% RSLogix 500 project TEMPLATE_BAK000.RSS, saved by version 8.30.00.16 %
PROJECT "UNTITLED"    % processor: Bul.1763 MicroLogix 1100 Series B %

PROGRAM FILES
  LAD 2 "MAIN"  10 rungs
  LAD 3 "DIGIT IN"  2 rungs
  LAD 4 "DIGIT OUT"  2 rungs
  LAD 5 "CTRL LOGIC"  5 rungs
  LAD 6 "HOA"  5 rungs
  LAD 7 "ANLG IN"  2 rungs
  LAD 8 "ANLG OUT"  1 rungs
  LAD 9 "ALARMS"  5 rungs
  LAD 10 "SYS MODES"  1 rungs
  LAD 11 "PROC LOGIC"  1 rungs

DATA FILES
  O0 OUTPUT  4 elements
  I1 INPUT  6 elements
  S2 STATUS  66 elements
  B3 BINARY  1 elements
  T4 TIMER  1 elements
  C5 COUNTER  1 elements
  R6 CONTROL  1 elements
  N7 INTEGER  1 elements
  F8 FLOAT  1 elements

LADDER 2 "MAIN"
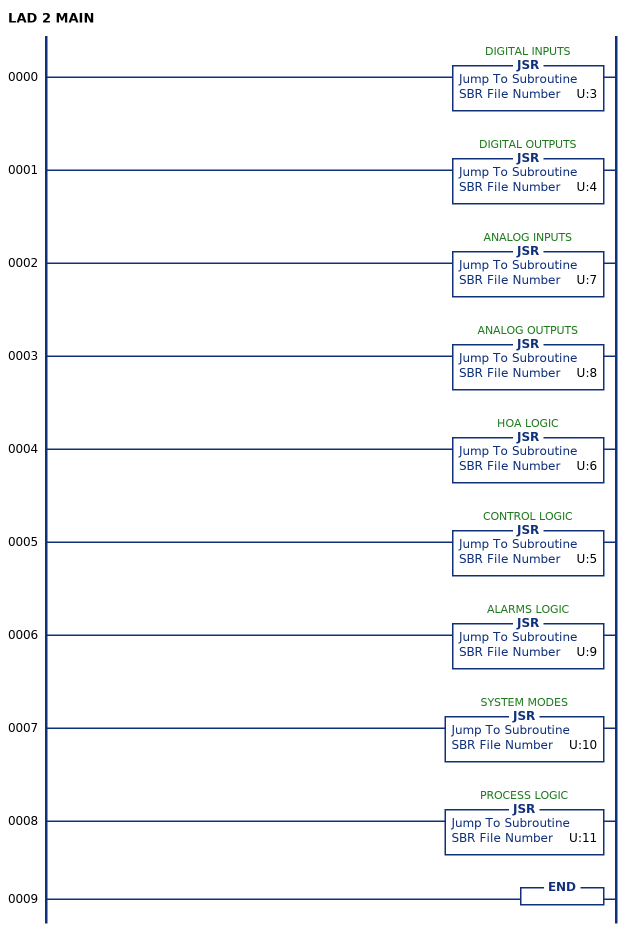
% Rung: 0 %
SOR JSR U:3 EOR
%   U:3  "DIGITAL INPUTS" %
% Rung: 1 %
SOR JSR U:4 EOR
%   U:4  "DIGITAL OUTPUTS" %
% Rung: 2 %
SOR JSR U:7 EOR
%   U:7  "ANALOG INPUTS" %
% Rung: 3 %
SOR JSR U:8 EOR
%   U:8  "ANALOG OUTPUTS" %
% Rung: 4 %
SOR JSR U:6 EOR
%   U:6  "HOA LOGIC" %
% Rung: 5 %
SOR JSR U:5 EOR
%   U:5  "CONTROL LOGIC" %
% Rung: 6 %
SOR JSR U:9 EOR
%   U:9  "ALARMS LOGIC" %
% Rung: 7 %
SOR JSR U:10 EOR
%   U:10  "SYSTEM MODES" %
% Rung: 8 %
SOR JSR U:11 EOR
%   U:11  "PROCESS LOGIC" %
% Rung: 9 %
SOR END EOR

LADDER 3 "DIGIT IN"
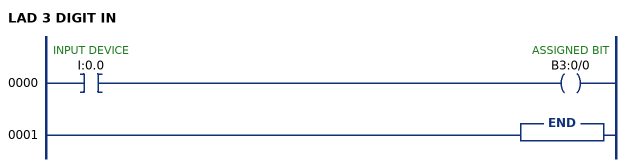
% Rung: 0 %  % edit flag set %
SOR XIC I:0.0 OTE B3:0/0 EOR
%   I:0.0  "INPUT DEVICE" %
%   B3:0/0  "ASSIGNED BIT" %
% Rung: 1 %
SOR END EOR

LADDER 4 "DIGIT OUT"
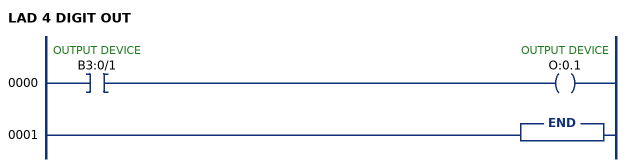
% Rung: 0 %  % edit flag set %
SOR XIC B3:0/1 OTE O:0.1 EOR
%   B3:0/1  "OUTPUT DEVICE" %
%   O:0.1  "OUTPUT DEVICE" %
% Rung: 1 %
SOR END EOR

LADDER 5 "CTRL LOGIC"
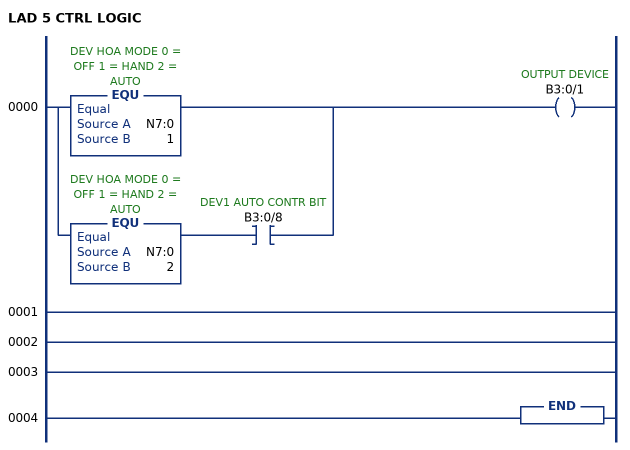
% Rung: 0 %  % edit flag set %
SOR BST EQU N7:0 1 NXB EQU N7:0 2 XIC B3:0/8 BND OTE B3:0/1 EOR
%   N7:0  "DEV HOA MODE 0 = OFF 1 = HAND 2 = AUTO" %
%   B3:0/8  "DEV1 AUTO CONTR BIT" %
%   B3:0/1  "OUTPUT DEVICE" %
% Rung: 1 %  % edit flag set %
SOR EOR
% Rung: 2 %  % edit flag set %
SOR EOR
% Rung: 3 %  % edit flag set %
SOR EOR
% Rung: 4 %
SOR END EOR

LADDER 6 "HOA"
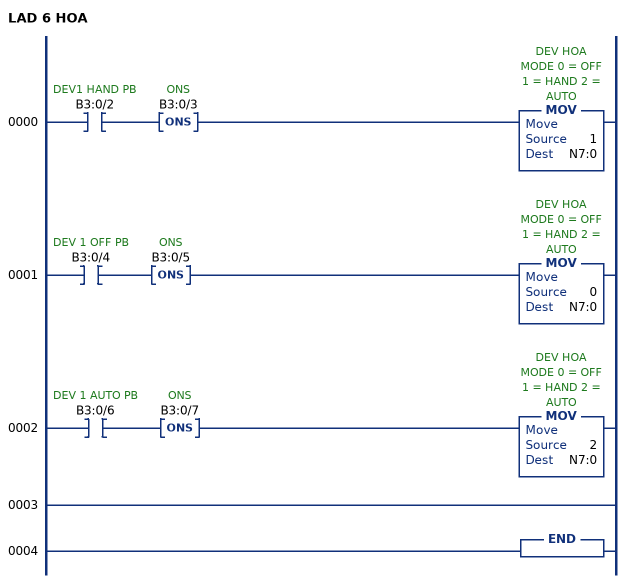
% Rung: 0 %  % edit flag set %
SOR XIC B3:0/2 ONS B3:0/3 MOV 1 N7:0 EOR
%   B3:0/2  "DEV1 HAND PB" %
%   B3:0/3  "ONS" %
%   N7:0  "DEV HOA MODE 0 = OFF 1 = HAND 2 = AUTO" %
% Rung: 1 %  % edit flag set %
SOR XIC B3:0/4 ONS B3:0/5 MOV 0 N7:0 EOR
%   B3:0/4  "DEV 1 OFF PB" %
%   B3:0/5  "ONS" %
%   N7:0  "DEV HOA MODE 0 = OFF 1 = HAND 2 = AUTO" %
% Rung: 2 %  % edit flag set %
SOR XIC B3:0/6 ONS B3:0/7 MOV 2 N7:0 EOR
%   B3:0/6  "DEV 1 AUTO PB" %
%   B3:0/7  "ONS" %
%   N7:0  "DEV HOA MODE 0 = OFF 1 = HAND 2 = AUTO" %
% Rung: 3 %  % edit flag set %
SOR EOR
% Rung: 4 %
SOR END EOR

LADDER 7 "ANLG IN"
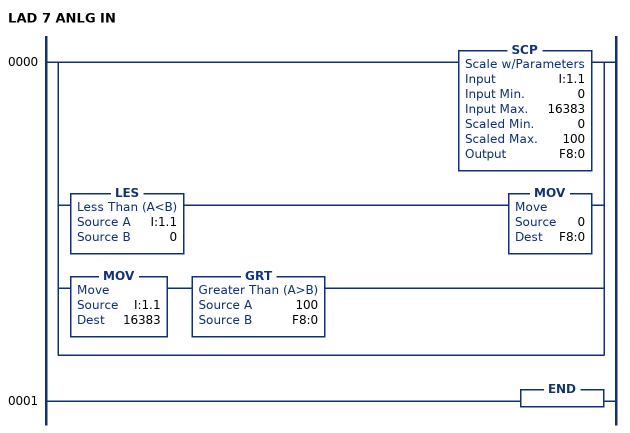
% Rung: 0 %  % edit flag set %
SOR BST SCP I:1.1 0 16383 0 100 F8:0 NXB LES I:1.1 0 MOV 0 F8:0 NXB MOV I:1.1 16383 GRT 100 F8:0 NXB BND EOR
% Rung: 1 %
SOR END EOR

LADDER 9 "ALARMS"
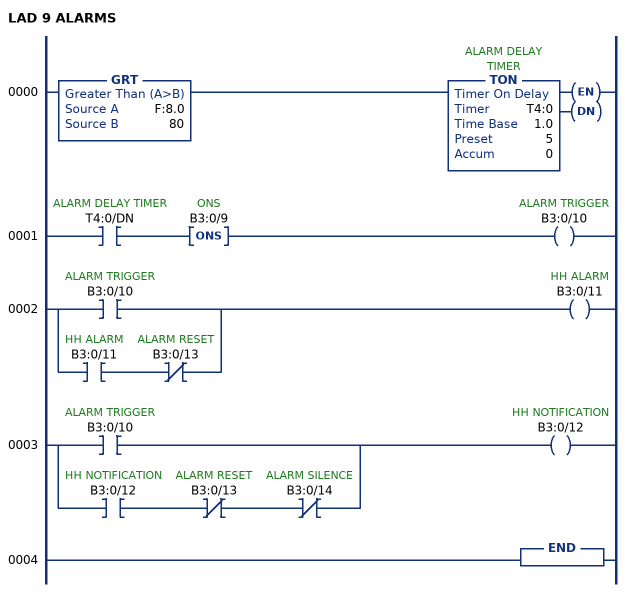
% Rung: 0 %  % edit flag set %
SOR GRT F:8.0 80 TON T4:0 1.0 5 0 EOR
%   T4:0  "ALARM DELAY TIMER" %
% Rung: 1 %  % edit flag set %
SOR XIC T4:0/DN ONS B3:0/9 OTE B3:0/10 EOR
%   T4:0  "ALARM DELAY TIMER" %
%   B3:0/9  "ONS" %
%   B3:0/10  "ALARM TRIGGER" %
% Rung: 2 %  % edit flag set %
SOR BST XIC B3:0/10 NXB XIC B3:0/11 XIO B3:0/13 BND OTE B3:0/11 EOR
%   B3:0/10  "ALARM TRIGGER" %
%   B3:0/11  "HH ALARM" %
%   B3:0/13  "ALARM RESET" %
% Rung: 3 %  % edit flag set %
SOR BST XIC B3:0/10 NXB XIC B3:0/12 XIO B3:0/13 XIO B3:0/14 BND OTE B3:0/12 EOR
%   B3:0/10  "ALARM TRIGGER" %
%   B3:0/12  "HH NOTIFICATION" %
%   B3:0/13  "ALARM RESET" %
%   B3:0/14  "ALARM SILENCE" %
% Rung: 4 %
SOR END EOR

OTHER DOCUMENTED ADDRESSES
  F8:8/0  "ANALOG INPUT VALUE"
  I:0.0/1  "OUTPUT DEVICE"
  N8:0  "ANALOG INPUT SCALED VALUE"
